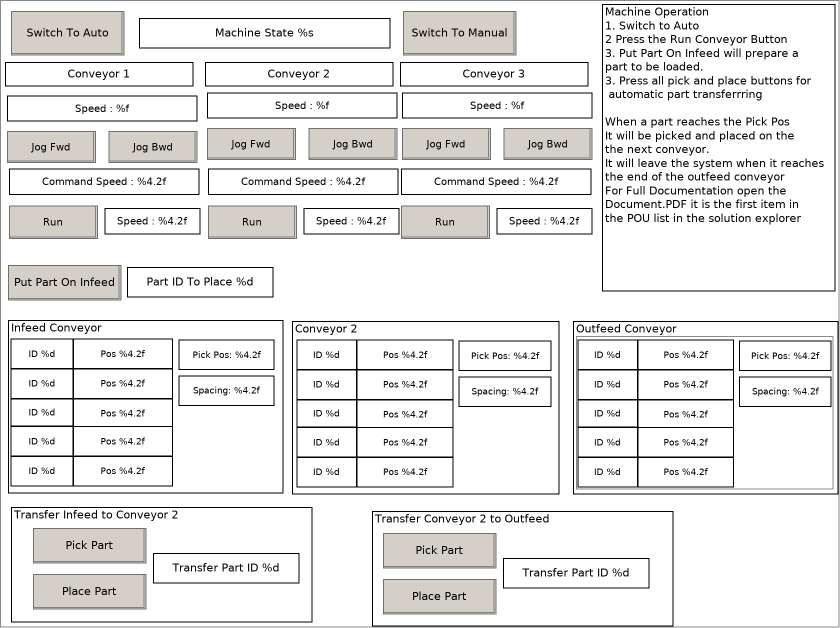
VISUALIZATION V_OOP_Conveyor  // 840x628
    Group (11,507 301x115)
        Rectangle (0,0 301x115), "Transfer Infeed to Conveyor 2"
        Button (22,21 113x35), "Pick Part", pressed state: MAIN.fbOOPConveyor.bPickPart
            toggle MAIN.fbOOPConveyor.bPickPart
        Rectangle (142,46 146x30), "Transfer Part ID %d", text variable: MAIN.fbOOPConveyor.fbTransfer1.stPart.iIDNumber
        Button (22,67 113x35), "Place Part", pressed state: MAIN.fbOOPConveyor.bPlacePart
            toggle MAIN.fbOOPConveyor.bPlacePart
    Button (11,11 113x44), "Switch To Auto"
        OnMouseDown: execute { MAIN.fbOOPConveyor.eMachineState := E_SwitchingToAuto; }
    Button (403,11 113x44), "Switch To Manual"
        OnMouseDown: execute { MAIN.fbOOPConveyor.eMachineState := E_SwitchingToManual; }
    Rectangle (139,18 251x30), "Machine State %s", text variable: MAIN.fbOOPConveyor.eMachineState
    Frame (10,99 189x66)
        shows Conveyor(bJogFwd := MAIN.fbOOPConveyor.bJogFwd, bJogBwd := MAIN.fbOOPConveyor.bJogBwd, fSpeed := MAIN.fbOOPConveyor.AxisRef[1].NcToPlc.ActVelo)
    Rectangle (5,62 188x24), "Conveyor 1"
    Frame (210,96 189x66)
        shows Conveyor(bJogFwd := MAIN.fbOOPConveyor.bJogFwd, bJogBwd := MAIN.fbOOPConveyor.bJogBwd, fSpeed := MAIN.fbOOPConveyor.iAnalogValue)
    Rectangle (205,62 188x24), "Conveyor 2"
    Frame (405,96 189x66)
        shows Conveyor(bJogFwd := MAIN.fbOOPConveyor.bJogFwd, bJogBwd := MAIN.fbOOPConveyor.bJogBwd, fSpeed := MAIN.fbOOPConveyor.AxisRef[2].NcToPlc.ActVelo)
    Rectangle (400,62 188x24), "Conveyor 3"
    Frame (11,174 191x67)
        shows ConveyorAuto(bRunConveyor := MAIN.fbOOPConveyor.bRunConveyor, fActualSpeed := MAIN.fbOOPConveyor.AxisRef[1].NcToPlc.ActVelo, fCmdSpeed := MAIN.fbOOPConveyor.fConveyorCmdSpeed)
    Button (8,265 113x35), "Put Part On Infeed", pressed state: MAIN.fbOOPConveyor.bPartPresent
        toggle MAIN.fbOOPConveyor.bPartPresent
    Frame (210,174 191x67)
        shows ConveyorAuto(bRunConveyor := MAIN.fbOOPConveyor.bRunConveyor, fActualSpeed := MAIN.fbOOPConveyor.fbConveyor2.fCurrentSpeed, fCmdSpeed := MAIN.fbOOPConveyor.fConveyorCmdSpeed)
    Rectangle (127,267 146x30), "Part ID To Place %d", text variable: arrParts[1].iIDNumber
    Group (292,321 267x173)
        Rectangle (0,0 267x173), "Conveyor 2"
        Frame (3,15 258x153)
            shows ConveyorData(fbConveyor := MAIN.fbOOPConveyor.fbConveyor2)
    Frame (403,174 191x67)
        shows ConveyorAuto(bRunConveyor := MAIN.fbOOPConveyor.bRunConveyor, fActualSpeed := MAIN.fbOOPConveyor.fbConveyor3.fCurrentSpeed, fCmdSpeed := MAIN.fbOOPConveyor.fConveyorCmdSpeed)
    Rectangle (8,320 275x173), "Infeed Conveyor"
    Frame (9,335 267x153)
        shows ConveyorData(fbConveyor := MAIN.fbOOPConveyor.fbInfeedConveyor)
    Group (372,511 301x115)
        Rectangle (0,0 301x115), "Transfer Conveyor 2 to Outfeed"
        Button (11,22 113x35), "Pick Part", pressed state: MAIN.fbOOPConveyor.bPickPart2
            toggle MAIN.fbOOPConveyor.bPickPart2
        Rectangle (131,47 146x30), "Transfer Part ID %d", text variable: MAIN.fbOOPConveyor.fbTransfer2.stPart.iIDNumber
        Button (11,68 113x35), "Place Part", pressed state: MAIN.fbOOPConveyor.bPlacePart2
            toggle MAIN.fbOOPConveyor.bPlacePart2
    Group (573,321 265x173)
        Rectangle (0,0 265x173), "Outfeed Conveyor"
        Frame (3,15 257x153)
            shows ConveyorData(fbConveyor := MAIN.fbOOPConveyor.fbConveyor3)
    Rectangle (602,4 233x287), "Machine Operation 1. Switch to Auto 2 Press the Run Conveyor Button 3. Put Part On Infeed will prepare a part to be loaded. 3. Press all pick and place buttons for automatic part transferrring When a part reaches the Pick Pos It will be picked and placed on the the next conveyor. It will leave the system when it reaches the end of the outfeed conveyor For Full Documentation open the Document.PDF it is the first item in the POU list in the solution explorer"
END_VISUALIZATION

// ---- POUs/Sample UML SC/Visu_Composite.TcVIS
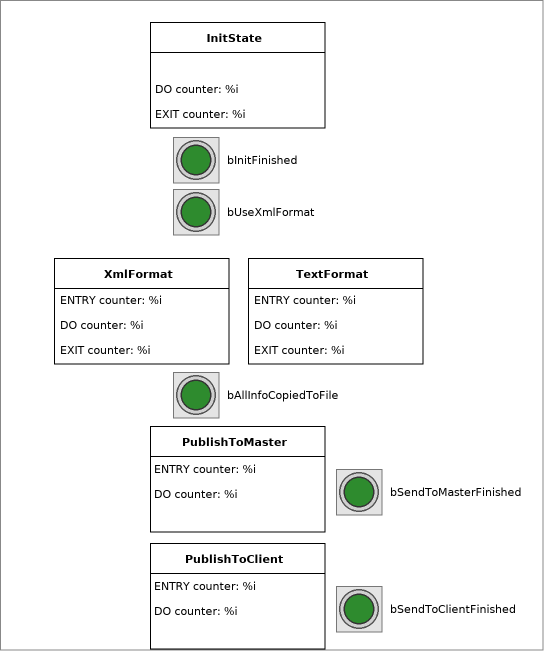
VISUALIZATION Visu_Composite  // 544x651
    Rectangle (150,22 175x106)
    Line (150,52) (325,52)
    Label (152,27 165x23), "InitState"
    Rectangle (54,258 175x106)
    Line (54,288) (229,288)
    Label (56,263 165x23), "XmlFormat"
    Rectangle (248,258 175x106)
    Line (248,288) (423,288)
    Label (250,263 165x23), "TextFormat"
    Rectangle (150,426 175x106)
    Line (150,456) (325,456)
    Label (152,431 165x23), "PublishToMaster"
    Rectangle (150,543 175x106)
    Line (150,573) (325,573)
    Label (152,548 165x23), "PublishToClient"
    PushSwitch (173,137 46x46), variable: MAIN.fbUmlSc.bInitFinished, behaviour: TOGGLE, style: Switch-PushSwitch-Green
    Label (224,149 118x23), "bInitFinished"
    PushSwitch (173,189 46x46), variable: MAIN.fbUmlSc.bUseXmlFormat, behaviour: TOGGLE, style: Switch-PushSwitch-Green
    Label (224,201 118x23), "bUseXmlFormat"
    PushSwitch (173,372 46x46), variable: MAIN.fbUmlSc.bAllInfoCopiedToFile, behaviour: TOGGLE, style: Switch-PushSwitch-Green
    Label (224,384 137x23), "bAllInfoCopiedToFile"
    PushSwitch (336,469 46x46), variable: MAIN.fbUmlSc.bSendToMasterFinished, behaviour: TOGGLE, style: Switch-PushSwitch-Green
    Label (387,481 155x23), "bSendToMasterFinished"
    PushSwitch (336,586 46x46), variable: MAIN.fbUmlSc.bSendToClientFinished, behaviour: TOGGLE, style: Switch-PushSwitch-Green
    Label (387,598 141x23), "bSendToClientFinished"
    Rectangle (152,54 169x21), text variable: GVL.nCounterInit
    Rectangle (152,79 169x21), "DO counter: %i", text variable: GVL.nCounterInit
    Rectangle (152,104 169x21), "EXIT counter: %i", text variable: GVL.nCounterSaveInitSettings
    Rectangle (57,290 169x21), "ENTRY counter: %i", text variable: GVL.nCounterClearXml
    Rectangle (57,315 169x21), "DO counter: %i", text variable: GVL.nCounterFillXml
    Rectangle (57,340 169x21), "EXIT counter: %i", text variable: GVL.nCounterSaveXml
    Rectangle (251,290 169x21), "ENTRY counter: %i", text variable: GVL.nCounterClearText
    Rectangle (251,315 169x21), "DO counter: %i", text variable: GVL.nCounterFillText
    Rectangle (251,340 169x21), "EXIT counter: %i", text variable: GVL.nCounterSaveText
    Rectangle (151,459 169x21), "ENTRY counter: %i", text variable: GVL.nCounterGetMasterID
    Rectangle (151,484 169x21), "DO counter: %i", text variable: GVL.nCounterSendToMaster
    Rectangle (151,509 169x21), text variable: GVL.nCounterInit
    Rectangle (151,576 169x21), "ENTRY counter: %i", text variable: GVL.nCounterGetClientID
    Rectangle (151,601 169x21), "DO counter: %i", text variable: GVL.nCounterSendToClient
    Rectangle (151,626 169x21), text variable: GVL.nCounterInit
END_VISUALIZATION

// ---- POUs/Sample UML SC/Visu_Lamp.TcVIS
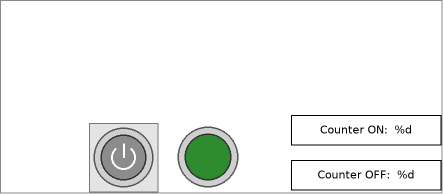
VISUALIZATION Visu_Lamp  // 443x194
    Lamp1 (173,122 70x70), variable: MAIN.fbUmlSc_Lamp.ObLamp, style: Lamp-Lamp1-Green
    PowerSwitch (69,123 109x69), variable: MAIN.fbUmlSc_Lamp.bPower, behaviour: TOGGLE, style: Switch-PowerSwitch-Gray
    Rectangle (291,115 150x30), "Counter ON: %d", text variable: MAIN.fbUmlSc_Lamp.nCounterOn
    Rectangle (291,160 150x30), "Counter OFF: %d", text variable: MAIN.fbUmlSc_Lamp.nCounterOff
END_VISUALIZATION

// ---- VISUs/MotionProfiles.TcVIS
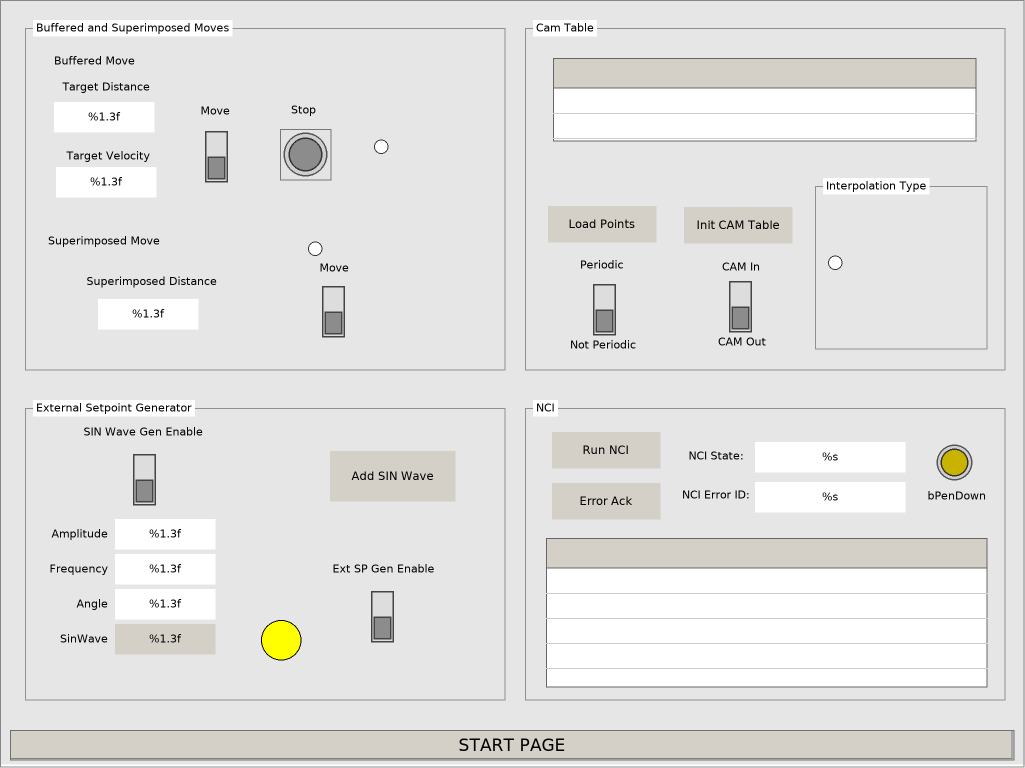
VISUALIZATION MotionProfiles  // 1025x768
    Rectangle (1,-4 1024x768)
    Button (10,730 1004x30), "START PAGE"
        OnMouseClick: change screen: HmiStartPage
    GroupBox (25,20 480x350), "Buffered and Superimposed Moves"
        Ellipse (236,600 40x40), colour toggle: Ext_SP_Gen.bAddSin
            toggle Ext_SP_Gen.bAddSin
        Label (12,30 115x22), "Buffered Move"
        Rectangle (29,82 100x30), "%1.3f", text variable: Axis3.lrMstrTarg2
            OnMouseDown: write the text variable via VisuDialogs.Numpad
        Rectangle (31,147 100x30), "%1.3f", text variable: Axis3.lrMstrVelo2
            OnMouseDown: write the text variable via VisuDialogs.Numpad
        Rectangle (30,56 98x22), "Target Distance"
        Rectangle (30,125 98x22), "Target Velocity"
        DipSwitch (166,108 51x57), variable: Axis3.bMvMstr2, behaviour: TOGGLE, style: Switch-DipSwitch-Gray
        RadioButton (347,95 96x63), variable: Axis3.iMstrMvMode2
            Areas[0]: Text=Absolute
            Areas[1]: Text=Relative
        PushSwitch (255,106 51x57), variable: Axis3.bStop, behaviour: TOGGLE, style: Switch-PushSwitch-Gray
        Label (12,210 134x22), "Superimposed Move"
        Label (159,80 63x22), "Move"
        Label (247,79 63x22), "Stop"
        Rectangle (73,279 100x30), "%1.3f", text variable: Axis3.lrMstrTarg3
            OnMouseDown: write the text variable via VisuDialogs.Numpad
        Rectangle (53,251 142x21), "Superimposed Distance"
        DipSwitch (283,263 51x57), variable: Axis3.bMvMstr2, behaviour: TOGGLE, style: Switch-DipSwitch-Gray
        Label (278,237 63x22), "Move"
    GroupBox (25,400 480x300), "External Setpoint Generator"
        DipSwitch (94,51 51x57), variable: Ext_SP_Gen.bSinGen, behaviour: TOGGLE, style: Switch-DipSwitch-Gray
        Label (45,21 147x22), "SIN Wave Gen Enable"
        DipSwitch (332,188 51x57), variable: Ext_SP_Gen.bMstrExtSP, behaviour: TOGGLE, style: Switch-DipSwitch-Gray
        Label (285,154 147x30), "Ext SP Gen Enable"
        Rectangle (11,158 75x22), "Frequency"
        Rectangle (305,51 125x50), "Add SIN Wave", colour toggle: Ext_SP_Gen.bAddSin
            toggle Ext_SP_Gen.bAddSin p2164770859=TRUE
    GroupBox (525,400 480x300), "NCI"
        Table (21,138 441x149), data array: NCI.aGCodeLines
            p3854506369: NCI.aGCodeLines[INDEX]
            p2232123230: Last 5 executed Gcode blocks
        Label (150,41 82x30), "NCI State:"
        Lamp1 (409,41 41x43), variable: NCI.bPenDown, style: Lamp-Lamp1-Yellow
        Rectangle (230,42 150x30), "%s", text variable: NCI.nNCI_State
        Label (150,80 82x30), "NCI Error ID:"
        Rectangle (230,82 150x30), "%s", text variable: NCI.nNciErrId
        Rectangle (27,32 108x36), "Run NCI", colour toggle: bRevSeqStart
            tap NCI.bRunNCI
        Rectangle (27,83 108x36), "Error Ack", colour toggle: bRevSeqStart
            tap NCI.bErrorAck
        Label (386,80 92x32), "bPenDown"
    GroupBox (525,20 480x350), "Cam Table"
        Rectangle (23,186 108x36), "Load Points", colour toggle: bRevSeqStart
            tap CamTable.bLoadPoints
        Rectangle (159,187 108x36), "Init CAM Table", colour toggle: bRevSeqStart
            tap CamTable.bCamInit
        DipSwitch (190,258 51x57), variable: CamTable.bCamIn, behaviour: TOGGLE, style: Switch-DipSwitch-Gray
        DipSwitch (54,261 51x57), variable: CamTable.bPeriodic, input disabled if: CamTable.bCamIn, behaviour: TOGGLE, style: Switch-DipSwitch-Gray
        Rectangle (168,311 98x22), "CAM Out"
        Rectangle (167,236 98x22), "CAM In"
        Rectangle (29,314 98x22), "Not Periodic"
        Rectangle (28,234 98x22), "Periodic"
        Table (28,38 423x83), data array: CamTable.arCamTable
            p3854506369: CamTable.arCamTable[0,INDEX]
            p1892666644: CamTable.arCamTable[1,INDEX]
            p338671338: CamTable.arCamTable[2,INDEX]
            p2170511999: CamTable.arCamTable[3,INDEX]
            p3723444502: CamTable.arCamTable[4,INDEX]
            p1218418051: CamTable.arCamTable[5,INDEX]
            p746581629: CamMotnFns.CamMotnFnPts[INDEX].SlavePos
            p3104783080: CamMotnFns.CamMotnFnPts[INDEX].SlaveVelo
            p2501879983: CamMotnFns.CamMotnFnPts[INDEX].SlaveAcc
            p7306298: CamMotnFns.CamMotnFnPts[INDEX].SlaveJerk
            p1137915858: CamTable.iSelY
            p1420305297: CamTable.iSelX
        GroupBox (290,158 172x171), "Interpolation Type"
            RadioButton (-509,19 137x103), variable: CamTable.iInterpType, input disabled if: CamTable.bCamIn
                Areas[0]: Text=Linear
                Areas[1]: Text=Spline
                Areas[2]: Text=Sliding Spline
        RadioButton (301,184 150x117), variable: CamTable.iInterpType, input disabled if: CamTable.bCamIn
            Areas[0]: Text=Linear
            Areas[1]: Text=Spline
            Areas[2]: Text=Sliding Spline
    Rectangle (115,624 100x30), "%1.3f", text variable: Ext_SP_Gen.lrSinWave
    Rectangle (115,589 100x30), "%1.3f", text variable: Ext_SP_Gen.rDeg
        OnMouseDown: write the text variable via VisuDialogs.Numpad
    Rectangle (58,593 53x22), "Angle"
    Rectangle (37,628 74x22), "SinWave"
    Rectangle (115,519 100x30), "%1.3f", text variable: Ext_SP_Gen.rSinAmp
        OnMouseDown: write the text variable via VisuDialogs.Numpad
    Rectangle (38,523 73x22), "Amplitude"
    Rectangle (115,554 100x30), "%1.3f", text variable: Ext_SP_Gen.rDegStep
        OnMouseDown: write the text variable via VisuDialogs.Numpad
END_VISUALIZATION

// ---- VISUs/HmiEtherCatDiagnostic.TcVIS
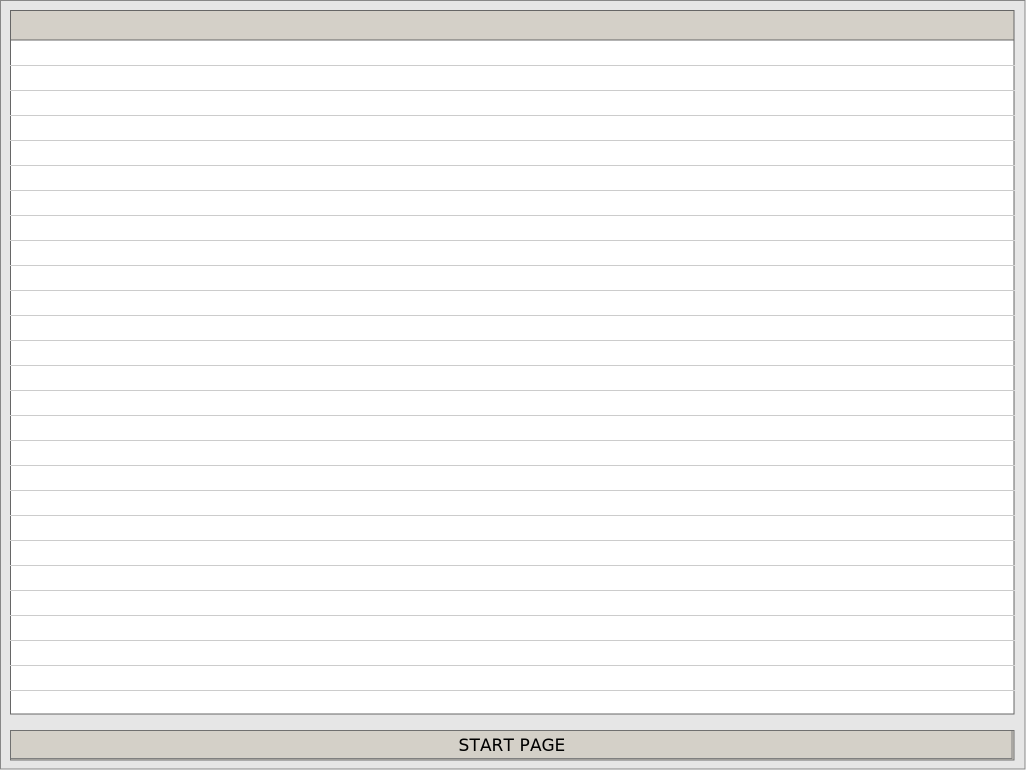
VISUALIZATION HmiEtherCatDiagnostic  // 1026x770
    Rectangle (0,0 1024x768)
    Button (10,730 1004x30), "START PAGE"
        OnMouseClick: change screen: HmiStartPage
    Table (10,10 1004x704), data array: fbDiagnosticEtherCAT.stEcTerminalDiagInfo
        p3854506369: fbDiagnosticEtherCAT.stEcTerminalDiagInfo[INDEX].nAddr
        p1892666644: fbDiagnosticEtherCAT.stEcTerminalDiagInfo[INDEX].sType
        p338671338: fbDiagnosticEtherCAT.stEcTerminalDiagInfo[INDEX].sName
        p2170511999: fbDiagnosticEtherCAT.stEcTerminalDiagInfo[INDEX].sTerminalStatus
END_VISUALIZATION

// ---- VISUs/HmiAxisReversingSequence.TcVIS
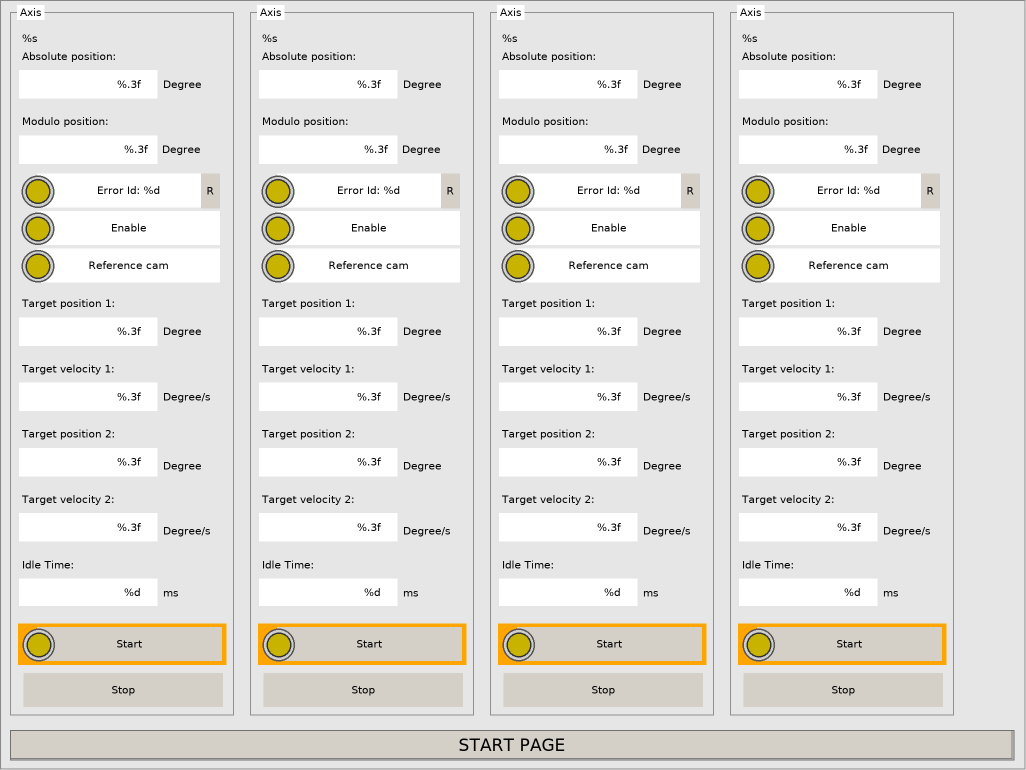
VISUALIZATION HmiAxisReversingSequence  // 1026x770
    Rectangle (0,0 1024x768)
    Button (10,730 1004x30), "START PAGE"
        OnMouseClick: change screen: HmiStartPage
    Frame (10,5 230x710)
        shows TplAxisReversingSequence(sAxisDescription := Axis1.sAxisDescription, fAbsolutePositon := stAxis1.NcToPlc.ActPos, fModuloPositon := stAxis1.NcToPlc.ModuloActPos, bError := Axis1.bAxisErr, nErrorId := Axis1.nAxisErrId, bReset := Axis1.bReset, bPowerStatus := Axis1.fbAxis.bPowerStatus, bReferenceCam := bStepperReferenceCam, bRevSeqStart := Axis1.bRevSeqStart, bRevSeqStop := Axis1.fbAxis.bRevSeqStop, fRevSeqTargetPos1 := Axis1.fbAxis.fRevSeqTargetPos1, fRevSeqTargetVelo1 := Axis1.fbAxis.fRevSeqTargetVelo1, fRevSeqTargetPos2 := Axis1.fbAxis.fRevSeqTargetPos2, fRevSeqTargetVelo2 := Axis1.fbAxis.fRevSeqTargetVelo2, nRevSeqIdleTime := Axis1.fbAxis.nRevSeqIdleTime, bRevSeqDone := Axis1.fbAxis.bRevSeqDone, bRevSeqBusy := Axis1.fbAxis.bRevSeqBusy)
    Frame (250,5 230x710)
        shows TplAxisReversingSequence(sAxisDescription := Axis2.sAxisDescription, fAbsolutePositon := stAxis2.NcToPlc.ActPos, fModuloPositon := stAxis2.NcToPlc.ModuloActPos, bError := Axis2.bAxisErr, nErrorId := Axis2.nAxisErrId, bReset := Axis2.bReset, bPowerStatus := Axis2.fbAxis.bPowerStatus, bReferenceCam := bAxis2ReferenceCamEL7, bRevSeqStart := Axis2.bRevSeqStart, bRevSeqStop := Axis2.fbAxis.bRevSeqStop, fRevSeqTargetPos1 := Axis2.fbAxis.fRevSeqTargetPos1, fRevSeqTargetVelo1 := Axis2.fbAxis.fRevSeqTargetVelo1, fRevSeqTargetPos2 := Axis2.fbAxis.fRevSeqTargetPos2, fRevSeqTargetVelo2 := Axis2.fbAxis.fRevSeqTargetVelo2, nRevSeqIdleTime := Axis2.fbAxis.nRevSeqIdleTime, bRevSeqDone := Axis2.fbAxis.bRevSeqDone, bRevSeqBusy := Axis2.fbAxis.bRevSeqBusy)
    Frame (490,5 230x710)
        shows TplAxisReversingSequence(sAxisDescription := Axis3.sAxisDescription, fAbsolutePositon := stAxis3.NcToPlc.ActPos, fModuloPositon := stAxis3.NcToPlc.ModuloActPos, bError := Axis3.bAxisErr, nErrorId := Axis3.nAxisErrId, bReset := Axis3.bReset, bPowerStatus := Axis3.fbAxis.bPowerStatus, bReferenceCam := AxisGeneral.bAxis3ReferenceCam, bRevSeqStart := Axis3.bRevSeqStart, bRevSeqStop := Axis3.fbAxis.bRevSeqStop, fRevSeqTargetPos1 := Axis3.fbAxis.fRevSeqTargetPos1, fRevSeqTargetVelo1 := Axis3.fbAxis.fRevSeqTargetVelo1, fRevSeqTargetPos2 := Axis3.fbAxis.fRevSeqTargetPos2, fRevSeqTargetVelo2 := Axis3.fbAxis.fRevSeqTargetVelo2, nRevSeqIdleTime := Axis3.fbAxis.nRevSeqIdleTime, bRevSeqDone := Axis3.fbAxis.bRevSeqDone, bRevSeqBusy := Axis3.fbAxis.bRevSeqBusy)
    Frame (730,5 230x710)
        shows TplAxisReversingSequence(sAxisDescription := Axis4.sAxisDescription, fAbsolutePositon := stAxis4.NcToPlc.ActPos, fModuloPositon := stAxis4.NcToPlc.ModuloActPos, bError := Axis4.bAxisErr, nErrorId := Axis4.nAxisErrId, bReset := Axis4.bReset, bPowerStatus := Axis4.fbAxis.bPowerStatus, bReferenceCam := AxisGeneral.bAxis4ReferenceCam, bRevSeqStart := Axis4.bRevSeqStart, bRevSeqStop := Axis4.fbAxis.bRevSeqStop, fRevSeqTargetPos1 := Axis4.fbAxis.fRevSeqTargetPos1, fRevSeqTargetVelo1 := Axis4.fbAxis.fRevSeqTargetVelo1, fRevSeqTargetPos2 := Axis4.fbAxis.fRevSeqTargetPos2, fRevSeqTargetVelo2 := Axis4.fbAxis.fRevSeqTargetVelo2, nRevSeqIdleTime := Axis4.fbAxis.nRevSeqIdleTime, bRevSeqDone := Axis4.fbAxis.bRevSeqDone, bRevSeqBusy := Axis4.fbAxis.bRevSeqBusy)
END_VISUALIZATION

// ---- VISUs/HmiStartPage.TcVIS
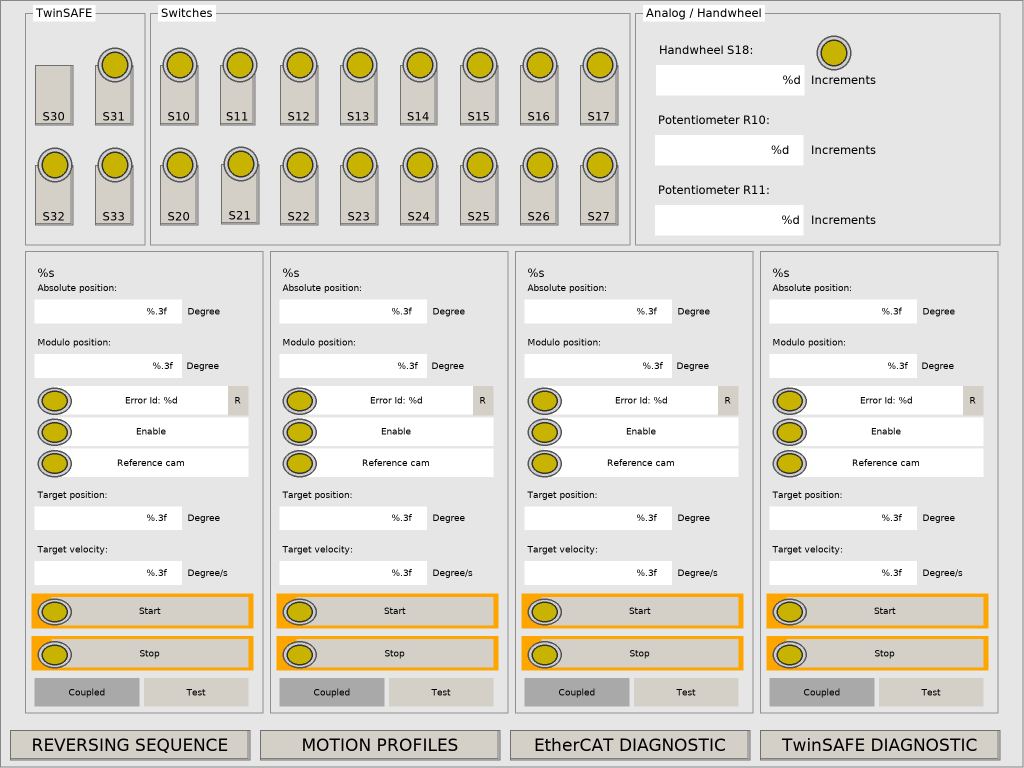
VISUALIZATION HmiStartPage  // 1024x768
    Rectangle (0,0 1024x768)
    Button (760,730 240x30), "TwinSAFE DIAGNOSTIC"
        OnMouseClick: change screen: HmiTwinSAFEDiagnostic
    Button (510,730 240x30), "EtherCAT DIAGNOSTIC"
        OnMouseClick: change screen: HmiEtherCatDiagnostic
    GroupBox (25,5 120x240), "TwinSAFE"
        Button (10,60 38x60), "S30", colour toggle: NOT TwinSAFE.fbSafeConnectionEL1904_1_Group1.bChannel1 and NOT TwinSAFE.fbSafeConnectionEL1904_1_Group1.bChannel2
            toggle bSwitchS31
        Button (70,60 38x60), "S31", colour toggle: bSwitchS31
            toggle bSwitchS31
        Lamp1 (70,40 40x40), variable: bLedH31, style: Lamp-Lamp1-Yellow
        Button (70,160 38x60), "S33", colour toggle: NOT TwinSAFE.fbSafeConnectionEL1904_2_Group1.bChannel3 and TwinSAFE.fbSafeConnectionEL1904_2_Group1.bChannel4
            toggle bSwitchS31
        Lamp1 (70,140 40x40), variable: bLedH33, style: Lamp-Lamp1-Yellow
        Button (10,160 38x60), "S32", colour toggle: NOT TwinSAFE.fbSafeConnectionEL1904_2_Group1.bChannel1 and NOT TwinSAFE.fbSafeConnectionEL1904_2_Group1.bChannel2
            toggle bSwitchS31
        Lamp1 (10,140 40x40), variable: bLedH32, style: Lamp-Lamp1-Yellow
    GroupBox (150,5 480x240), "Switches"
        Button (10,60 38x60), "S10", colour toggle: bSwitchS10
            toggle bSwitchS10
        Lamp1 (10,40 40x40), variable: bLedH10, style: Lamp-Lamp1-Yellow
        Button (70,60 35x60), "S11", colour toggle: bSwitchS11
            toggle bSwitchS11
        Lamp1 (70,40 40x40), variable: bLedH11, style: Lamp-Lamp1-Yellow
        Button (130,60 38x60), "S12", colour toggle: bSwitchS12
            toggle bSwitchS12
        Lamp1 (130,40 40x40), variable: bLedH12, style: Lamp-Lamp1-Yellow
        Button (190,60 37x60), "S13", colour toggle: bSwitchS13
            toggle bSwitchS13
        Lamp1 (190,40 40x40), variable: bLedH13, style: Lamp-Lamp1-Yellow
        Button (250,60 37x60), "S14", colour toggle: bSwitchS14
            toggle bSwitchS14
        Lamp1 (250,40 40x40), variable: bLedH14, style: Lamp-Lamp1-Yellow
        Button (310,60 38x60), "S15", colour toggle: bSwitchS15
            toggle bSwitchS15
        Lamp1 (310,40 40x40), variable: bLedH15, style: Lamp-Lamp1-Yellow
        Button (370,60 38x60), "S16", colour toggle: bSwitchS16
            toggle bSwitchS16
        Lamp1 (370,40 40x40), variable: bLedH16, style: Lamp-Lamp1-Yellow
        Button (430,60 38x60), "S17", colour toggle: bSwitchS17
            toggle bSwitchS17
        Lamp1 (430,40 40x40), variable: bLedH17, style: Lamp-Lamp1-Yellow
        Button (10,160 38x60), "S20", colour toggle: bSwitchS20
            toggle bSwitchS20
        Lamp1 (10,140 40x40), variable: bLedH20, style: Lamp-Lamp1-Yellow
        Button (71,159 38x60), "S21", colour toggle: bSwitchS21
            toggle bSwitchS21
        Lamp1 (71,139 40x40), variable: bLedH21, style: Lamp-Lamp1-Yellow
        Button (130,160 38x60), "S22", colour toggle: bSwitchS22
            toggle bSwitchS22
        Lamp1 (130,140 40x40), variable: bLedH22, style: Lamp-Lamp1-Yellow
        Button (190,160 38x60), "S23", colour toggle: bSwitchS23
            toggle bSwitchS23
        Lamp1 (190,140 40x40), variable: bLedH23, style: Lamp-Lamp1-Yellow
        Button (250,160 38x60), "S24", colour toggle: bSwitchS24
            toggle bSwitchS24
        Lamp1 (250,140 40x40), variable: bLedH24, style: Lamp-Lamp1-Yellow
        Button (310,160 38x60), "S25", colour toggle: bSwitchS25
            toggle bSwitchS25
        Lamp1 (310,140 40x40), variable: bLedH25, style: Lamp-Lamp1-Yellow
        Button (370,160 38x60), "S26", colour toggle: nAX5203DigitalInputs.2
            toggle nAX5203DigitalInputs.2
        Lamp1 (370,140 40x40), variable: bLedH26, style: Lamp-Lamp1-Yellow
        Button (430,160 38x60), "S27", colour toggle: nAX5203DigitalInputs.3
            toggle nAX5203DigitalInputs.3
        Lamp1 (430,140 40x40), variable: nAX5203DigitalOutputs.7, style: Lamp-Lamp1-Yellow
    GroupBox (635,5 365x240), "Analog / Handwheel"
        Rectangle (20,200 148x30), "%d", text variable: aOsAnalogInR11[0]
            OnMouseClick: write the text variable via VisuDialogs.Numpad, min 0, max 32767
        Label (173,200 118x30), "Increments"
        Label (20,170 197x30), "Potentiometer R11:"
        Rectangle (20,130 148x30), "%d", text variable: nAnalogInR10
            OnMouseClick: write the text variable via VisuDialogs.Numpad, min 0, max 32767
        Label (173,130 121x30), "Increments"
        Label (20,100 216x30), "Potentiometer R10:"
        Lamp1 (179,28 40x40), variable: bHandwheelSwitchS28, style: Lamp-Lamp1-Yellow
        Rectangle (21,60 148x30), "%d", text variable: nHandwheelCounter
            OnMouseClick: write the text variable via VisuDialogs.Numpad
        Label (173,60 133x30), "Increments"
        Label (21,30 216x30), "Handwheel S18:"
    Frame (25,245 240x470)
        shows TplAxisControl(sAxisDescription := Axis1.sAxisDescription, fAbsolutePositon := stAxis1.NcToPlc.ActPos, fModuloPositon := stAxis1.NcToPlc.ModuloActPos, bError := Axis1.bAxisErr, nErrorId := Axis1.nAxisErrId, bReset := Axis1.bReset, bPowerStatus := Axis1.fbAxis.bPowerStatus, bReferenceCam := bStepperReferenceCam, fMoveAbsPosition := Axis1.fMoveAbsPosition, fMoveAbsVelocity := Axis1.fMoveAbsVelocity, bStartMoveAbs := Axis1.bStartMoveAbs, bMoveAbsBusy := Axis1.bMoveAbsBusy, bMoveAbsDone := Axis1.bMoveAbsDone, bStop := Axis1.bStop, bStopBusy := Axis1.bStopAxisBusy, bStopDone := Axis1.bStopAxisDone, bAxisCoupled := Axis1.bAxisCoupled, bTestChangeTargetPosAxis := Axis1.bTestChangeTargetPos)
    Frame (270,245 240x470)
        shows TplAxisControl(sAxisDescription := Axis2.sAxisDescription, fAbsolutePositon := stAxis2.NcToPlc.ActPos, fModuloPositon := stAxis2.NcToPlc.ModuloActPos, bError := Axis2.bAxisErr, nErrorId := Axis2.nAxisErrId, bReset := Axis2.bReset, bPowerStatus := Axis2.fbAxis.bPowerStatus, bReferenceCam := bAxis2ReferenceCamEL7, fMoveAbsPosition := Axis2.fMoveAbsPosition, fMoveAbsVelocity := Axis2.fMoveAbsVelocity, bStartMoveAbs := Axis2.bStartMoveAbs, bMoveAbsBusy := Axis2.bMoveAbsBusy, bMoveAbsDone := Axis2.bMoveAbsDone, bStop := Axis2.bStop, bStopBusy := Axis2.bStopAxisBusy, bStopDone := Axis2.bStopAxisDone, bAxisCoupled := Axis2.bAxisCoupled, bTestChangeTargetPosAxis := Axis2.bTestChangeTargetPos)
    Frame (515,245 240x470)
        shows TplAxisControl(sAxisDescription := Axis3.sAxisDescription, fAbsolutePositon := stAxis3.NcToPlc.ActPos, fModuloPositon := stAxis3.NcToPlc.ModuloActPos, bError := Axis3.bAxisErr, nErrorId := Axis3.nAxisErrId, bReset := Axis3.bReset, bPowerStatus := Axis3.fbAxis.bPowerStatus, bReferenceCam := AxisGeneral.bAxis3ReferenceCam, fMoveAbsPosition := Axis3.fMoveAbsPosition, fMoveAbsVelocity := Axis3.fMoveAbsVelocity, bStartMoveAbs := Axis3.bStartMoveAbs, bMoveAbsBusy := Axis3.bMoveAbsBusy, bMoveAbsDone := Axis3.bMoveAbsDone, bStop := Axis3.bStop, bStopBusy := Axis3.bStopAxisBusy, bStopDone := Axis3.bStopAxisDone, bAxisCoupled := Axis3.bAxisCoupled, bTestChangeTargetPosAxis := Axis3.bTestChangeTargetPos)
    Frame (760,245 240x470)
        shows TplAxisControl(sAxisDescription := Axis4.sAxisDescription, fAbsolutePositon := stAxis4.NcToPlc.ActPos, fModuloPositon := stAxis4.NcToPlc.ModuloActPos, bError := Axis4.bAxisErr, nErrorId := Axis4.nAxisErrId, bReset := Axis4.bReset, bPowerStatus := Axis4.fbAxis.bPowerStatus, bReferenceCam := AxisGeneral.bAxis4ReferenceCam, fMoveAbsPosition := Axis4.fMoveAbsPosition, fMoveAbsVelocity := Axis4.fMoveAbsVelocity, bStartMoveAbs := Axis4.bStartMoveAbs, bMoveAbsBusy := Axis4.bMoveAbsBusy, bMoveAbsDone := Axis4.bMoveAbsDone, bStop := Axis4.bStop, bStopBusy := Axis4.bStopAxisBusy, bStopDone := Axis4.bStopAxisDone, bAxisCoupled := Axis4.bAxisCoupled, bTestChangeTargetPosAxis := Axis4.bTestChangeTargetPos)
    Button (10,730 240x30), "REVERSING SEQUENCE"
        OnMouseClick: change screen: HmiAxisReversingSequence
    Button (260,730 240x30), "MOTION PROFILES"
        OnMouseClick: change screen: MotionProfiles
END_VISUALIZATION

// ---- VISUs/HmiTemplatesAxis/TplAxisControl.TcVIS
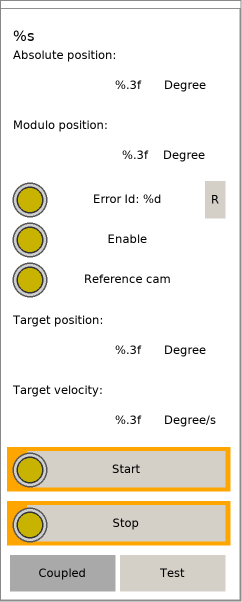
VISUALIZATION TplAxisControl  // 242x602
VAR_IN_OUT
	sAxisDescription				:STRING;
	fAbsolutePositon				:LREAL;
	fModuloPositon					:LREAL;
	bError							:BOOL;
	nErrorId						:DWORD;
	bReset							:BOOL;
	bPowerStatus					:BOOL;
	bReferenceCam					:BOOL;
	fMoveAbsPosition				:LREAL;
	fMoveAbsVelocity				:LREAL;
	bStartMoveAbs					:BOOL;
	bMoveAbsBusy					:BOOL;
	bMoveAbsDone					:BOOL;
	bStop							:BOOL;
	bStopBusy						:BOOL;
	bStopDone						:BOOL;
	bAxisCoupled					:BOOL;
	bTestChangeTargetPosAxis		:BOOL;
END_VAR
(* End *)
    GroupBox (0,0 240x600)
        Rectangle (7,501 223x44), invisible if: NOT bStopBusy
        Rectangle (7,447 223x44), invisible if: NOT bMoveAbsBusy
        Rectangle (27,451 198x36), "Start", colour toggle: bStartMoveAbs
            toggle bStartMoveAbs
        Group (10,110 230x60)
            Rectangle (0,30 148x30), "%.3f", text variable: fModuloPositon
            Label (150,30 80x30), "Degree"
            Label (0,0 200x30), "Modulo position:"
        Group (10,40 227x60)
            Rectangle (0,30 148x30), "%.3f", text variable: fAbsolutePositon
            Label (151,30 76x30), "Degree"
            Label (0,0 216x30), "Absolute position:"
        Group (10,180 200x40)
            Rectangle (20,1 195x36), "Error Id: %d", text variable: nErrorId
            Lamp1 (0,0 40x40), variable: bError, style: Lamp-Lamp1-Yellow
        Group (10,220 215x40)
            Rectangle (20,1 195x36), "Enable"
            Lamp1 (0,0 40x40), variable: bPowerStatus, style: Lamp-Lamp1-Yellow
        Group (10,260 215x40)
            Rectangle (20,1 195x36), "Reference cam"
            Lamp1 (0,0 40x40), variable: bReferenceCam, style: Lamp-Lamp1-Yellow
        Rectangle (205,181 20x37), "R", tooltip "Reset", colour toggle: bReset
            tap bReset
        Rectangle (27,505 198x36), "Stop", colour toggle: bStop
            toggle bStop
        Rectangle (10,555 105x36), "Coupled", colour toggle: bAxisCoupled
        Rectangle (10,25 230x22), "%s", text variable: sAxisDescription
        Rectangle (10,335 148x30), "%.3f", text variable: fMoveAbsPosition
            OnMouseClick: write the text variable via VisuDialogs.Numpad
        Label (161,335 76x30), "Degree"
        Label (10,305 216x30), "Target position:"
        Rectangle (10,405 148x30), "%.3f", text variable: fMoveAbsVelocity
            OnMouseClick: write the text variable via VisuDialogs.Numpad
        Label (161,405 76x30), "Degree/s"
        Label (10,375 216x30), "Target velocity:"
        Lamp1 (10,505 40x40), variable: bStopDone, style: Lamp-Lamp1-Yellow
        Rectangle (120,555 105x36), "Test", colour toggle: bTestChangeTargetPosAxis
            toggle bTestChangeTargetPosAxis
        Lamp1 (10,450 40x40), variable: bMoveAbsDone, style: Lamp-Lamp1-Yellow
END_VISUALIZATION

// ---- VISUs/HmiTemplatesAxis/TplAxisReversingSequence.TcVIS
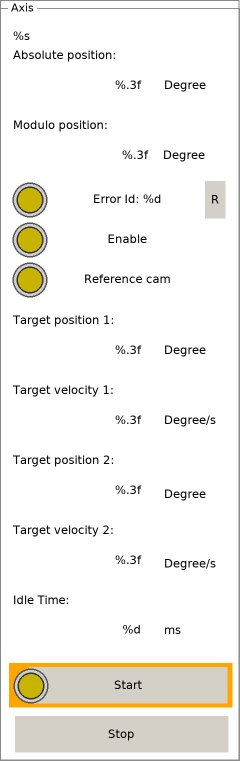
VISUALIZATION TplAxisReversingSequence  // 240x761
VAR_IN_OUT
	sAxisDescription				:STRING;
	fAbsolutePositon				:LREAL;
	fModuloPositon					:LREAL;
	bError							:BOOL;
	nErrorId						:DWORD;
	bReset							:BOOL;
	bPowerStatus					:BOOL;
	bReferenceCam					:BOOL;
	bRevSeqStart					:BOOL;
	bRevSeqStop						:BOOL;
	fRevSeqTargetPos1				:LREAL;
	fRevSeqTargetVelo1				:LREAL;
	fRevSeqTargetPos2				:LREAL;
	fRevSeqTargetVelo2				:LREAL;
	nRevSeqIdleTime					:UINT;
	bRevSeqDone						:BOOL;
	bRevSeqBusy						:BOOL;
END_VAR
    GroupBox (0,0 240x761), "Axis"
        Group (10,40 227x60)
            Rectangle (0,30 148x30), "%.3f", text variable: fAbsolutePositon
            Label (151,30 76x30), "Degree"
            Label (0,0 216x30), "Absolute position:"
        Group (10,180 200x40)
            Rectangle (20,1 195x36), "Error Id: %d", text variable: nErrorId
            Lamp1 (0,0 40x40), variable: bError, style: Lamp-Lamp1-Yellow
        Group (10,220 215x40)
            Rectangle (20,1 195x36), "Enable"
            Lamp1 (0,0 40x40), variable: bPowerStatus, style: Lamp-Lamp1-Yellow
        Group (10,260 215x40)
            Rectangle (20,1 195x36), "Reference cam"
            Lamp1 (0,0 40x40), variable: bReferenceCam, style: Lamp-Lamp1-Yellow
        Rectangle (205,181 20x37), "R", tooltip "Reset", colour toggle: bReset
            tap bReset
        Rectangle (10,25 230x22), "%s", text variable: sAxisDescription
        Rectangle (10,335 148x30), "%.3f", text variable: fRevSeqTargetPos1
            OnMouseClick: write the text variable via VisuDialogs.Numpad
        Label (161,335 76x30), "Degree"
        Label (10,305 216x30), "Target position 1:"
        Rectangle (10,405 148x30), "%.3f", text variable: fRevSeqTargetVelo1
            OnMouseClick: write the text variable via VisuDialogs.Numpad
        Label (161,405 76x30), "Degree/s"
        Group (10,110 230x60)
            Rectangle (0,30 148x30), "%.3f", text variable: fModuloPositon
            Label (150,30 80x30), "Degree"
            Label (0,0 200x30), "Modulo position:"
        Rectangle (9,663 223x44), invisible if: NOT bRevSeqBusy
        Rectangle (29,667 198x36), "Start", colour toggle: bRevSeqStart
            toggle bRevSeqStart
        Lamp1 (11,666 40x40), variable: bRevSeqDone, style: Lamp-Lamp1-Yellow
        Rectangle (15,716 213x36), "Stop", colour toggle: bRevSeqStop
            toggle bRevSeqStop
        Rectangle (10,615 148x29), "%d", text variable: nRevSeqIdleTime
            OnMouseClick: write the text variable via VisuDialogs.Numpad
        Label (10,585 216x30), "Idle Time:"
        Label (10,375 216x30), "Target velocity 1:"
    Label (161,479 76x30), "Degree"
    Rectangle (10,475 148x30), "%.3f", text variable: fRevSeqTargetPos2
        OnMouseClick: write the text variable via VisuDialogs.Numpad
    Label (10,445 216x30), "Target position 2:"
    Rectangle (10,545 148x30), "%.3f", text variable: fRevSeqTargetVelo2
        OnMouseClick: write the text variable via VisuDialogs.Numpad
    Label (161,549 76x29), "Degree/s"
    Label (10,515 216x30), "Target velocity 2:"
    Label (161,615 76x30), "ms"
END_VISUALIZATION

// ---- VISUs/HmiTemplatesTwinSAFE/TplTsConnectionAX5805.TcVIS
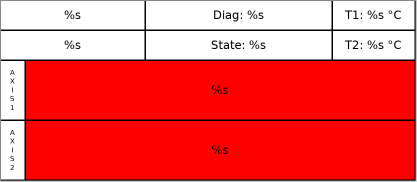
VISUALIZATION TplTsConnectionAX5805  // 417x182
VAR_IN_OUT
	stConnectionDiag 			:FB_TwinSafeConnectionAX5805;
END_VAR
(* End *)
    Rectangle (0,0 145x30), "%s", text variable: stConnectionDiag.sEcSlaveName
    Rectangle (25,60 49x30), "S-STO", colour toggle: stConnectionDiag.stSignalStatusMC1.bSafeTorqueOff_STO
    Rectangle (74,60 49x30), "S-SMM1", colour toggle: stConnectionDiag.stSignalStatusMC1.bSafeSpeedMonitor_SSM_1
    Rectangle (123,60 49x30), "S-SSM2", colour toggle: stConnectionDiag.stSignalStatusMC1.bSafeSpeedMonitor_SSM_2
    Rectangle (172,60 48x30), "S-SOS1", colour toggle: stConnectionDiag.stSignalStatusMC1.bSafeOperatingStop_SOS_1
    Rectangle (145,0 187x30), "Diag: %s", text variable: stConnectionDiag.sDiag, colour toggle: stConnectionDiag.sDiag <> 'No error'
    Rectangle (145,30 187x30), "State: %s", text variable: stConnectionDiag.sState
    Rectangle (0,30 145x30), "%s", text variable: stConnectionDiag.sEcSlaveType
    Rectangle (220,60 49x30), "S-SSR1", colour toggle: stConnectionDiag.stSignalStatusMC1.bSafeSpeedRange_SSR_1
    Rectangle (269,60 49x30), "S-SDIp", colour toggle: stConnectionDiag.stSignalStatusMC1.bSafeDirectionPositive_SDIp
    Rectangle (318,60 49x30), "S-SDIn", colour toggle: stConnectionDiag.stSignalStatusMC1.bSafeDirectionNegative_SDIn
    Rectangle (367,60 48x30), "S-Err Ack", colour toggle: stConnectionDiag.stSignalStatusMC1.bErrorAcknowledge_ErrAck
    Rectangle (25,90 49x30), "C-STO", colour toggle: stConnectionDiag.stSignalControlStatusMC1.bSafeTorqueOff_STO
    Rectangle (74,90 49x30), "C-SS1", colour toggle: stConnectionDiag.stSignalControlStatusMC1.bSafeStop1_SS1_1
    Rectangle (123,90 49x30), "C-SS2", colour toggle: stConnectionDiag.stSignalControlStatusMC1.bSafeStop2_SS2_1
    Rectangle (172,90 48x30), "C-SOS1", colour toggle: stConnectionDiag.stSignalControlStatusMC1.bSafeOperatingStop_SOS_1
    Rectangle (220,90 49x30), "C-SSR1", colour toggle: stConnectionDiag.stSignalControlStatusMC1.bSafeSpeedRange_SSR_1
    Rectangle (269,90 49x30), "C-SDIp", colour toggle: stConnectionDiag.stSignalControlStatusMC1.bSafeDirectionPositive_SDIp
    Rectangle (318,90 49x30), "C-SDIn", colour toggle: stConnectionDiag.stSignalControlStatusMC1.bSafeDirectionNegative_SDIn
    Rectangle (367,90 48x30), "C-Err Ack", colour toggle: stConnectionDiag.stSignalControlStatusMC1.bErrorAcknowledge_ErrAck
    Rectangle (332,0 83x30), "T1: %s °C", text variable: stConnectionDiag.stSlaveTemp.nInternalTemperature1, colour toggle: stConnectionDiag.bTempWarning
    Rectangle (332,30 83x30), "T2: %s °C", text variable: stConnectionDiag.stSlaveTemp.nInternalTemperature2, colour toggle: stConnectionDiag.bTempWarning
    Rectangle (25,120 49x30), "S-STO", colour toggle: stConnectionDiag.stSignalStatusMC2.bSafeTorqueOff_STO
    Rectangle (74,120 49x30), "S-SMM1", colour toggle: stConnectionDiag.stSignalStatusMC2.bSafeSpeedMonitor_SSM_1
    Rectangle (123,120 49x30), "S-SSM2", colour toggle: stConnectionDiag.stSignalStatusMC2.bSafeSpeedMonitor_SSM_2
    Rectangle (172,120 48x30), "S-SOS1", colour toggle: stConnectionDiag.stSignalStatusMC2.bSafeOperatingStop_SOS_1
    Rectangle (220,120 49x30), "S-SSR1", colour toggle: stConnectionDiag.stSignalStatusMC2.bSafeSpeedRange_SSR_1
    Rectangle (269,120 49x30), "S-SDIp", colour toggle: stConnectionDiag.stSignalStatusMC2.bSafeDirectionPositive_SDIp
    Rectangle (318,120 49x30), "S-SDIn", colour toggle: stConnectionDiag.stSignalStatusMC2.bSafeDirectionNegative_SDIn
    Rectangle (367,120 48x30), "S-Err Ack", colour toggle: stConnectionDiag.stSignalStatusMC2.bErrorAcknowledge_ErrAck
    Rectangle (25,150 49x30), "C-STO", colour toggle: stConnectionDiag.stSignalControlStatusMC2.bSafeTorqueOff_STO
    Rectangle (74,150 49x30), "C-SS1", colour toggle: stConnectionDiag.stSignalControlStatusMC2.bSafeStop1_SS1_1
    Rectangle (123,150 49x30), "C-SS2", colour toggle: stConnectionDiag.stSignalControlStatusMC2.bSafeStop2_SS2_1
    Rectangle (172,150 48x30), "C-SOS1", colour toggle: stConnectionDiag.stSignalControlStatusMC2.bSafeOperatingStop_SOS_1
    Rectangle (220,150 49x30), "C-SSR1", colour toggle: stConnectionDiag.stSignalControlStatusMC2.bSafeSpeedRange_SSR_1
    Rectangle (269,150 49x30), "C-SDIp", colour toggle: stConnectionDiag.stSignalControlStatusMC2.bSafeDirectionPositive_SDIp
    Rectangle (318,150 49x30), "C-SDIn", colour toggle: stConnectionDiag.stSignalControlStatusMC2.bSafeDirectionNegative_SDIn
    Rectangle (367,150 48x30), "C-Err Ack", colour toggle: stConnectionDiag.stSignalControlStatusMC2.bErrorAcknowledge_ErrAck
    Rectangle (0,60 25x60), "A X I S 1"
    Rectangle (0,120 25x60), "A X I S 2"
    Rectangle (26,61 388x58), "%s", text variable: stConnectionDiag.eErrIndicesFA82DiagnosisMC1, invisible if: NOT stConnectionDiag.bErrIndicesFA82DiagnosisMC1Err
    Rectangle (26,121 388x58), "%s", text variable: stConnectionDiag.eErrIndicesFA82DiagnosisMC2, invisible if: NOT stConnectionDiag.bErrIndicesFA82DiagnosisMC2Err
END_VISUALIZATION

// ---- VISUs/HmiTemplatesTwinSAFE/TplTsConnectionEK1914.TcVIS
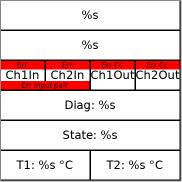
VISUALIZATION TplTsConnectionEK1914  // 182x182
VAR_IN_OUT
	stConnectionDiag 			:FB_TwinSafeConnectionEK1914;
END_VAR
(* End *)
    Rectangle (0,0 180x30), "%s", text variable: stConnectionDiag.sEcSlaveName, colour toggle: stConnectionDiag.sDiag = 'No error'
    Rectangle (0,60 45x30), "Ch1In", colour toggle: stConnectionDiag.bChannel1In
    Rectangle (45,60 45x30), "Ch2In", colour toggle: stConnectionDiag.bChannel2In
    Rectangle (90,60 45x30), "Ch1Out", colour toggle: stConnectionDiag.bChannel1Out
    Rectangle (135,60 45x30), "Ch2Out", colour toggle: stConnectionDiag.bChannel2Out
    Rectangle (0,90 180x30), "Diag: %s", text variable: stConnectionDiag.sDiag, colour toggle: stConnectionDiag.sDiag <> 'No error'
    Rectangle (0,120 180x30), "State: %s", text variable: stConnectionDiag.sState
    Rectangle (0,150 90x30), "T1: %s °C", text variable: stConnectionDiag.stSlaveTemp.nInternalTemperature1, colour toggle: stConnectionDiag.bTempWarning
    Rectangle (90,150 90x30), "T2: %s °C", text variable: stConnectionDiag.stSlaveTemp.nInternalTemperature2, colour toggle: stConnectionDiag.bTempWarning
    Rectangle (0,30 180x30), "%s", text variable: stConnectionDiag.sEcSlaveType
    Rectangle (1,61 43x8), "Err", invisible if: NOT stConnectionDiag.stTsDiagObjectsBitsEK1914.bErrInput1
    Rectangle (46,61 43x8), "Err", invisible if: NOT stConnectionDiag.stTsDiagObjectsBitsEK1914.bErrInput2
    Rectangle (91,61 43x8), "Err Cc", invisible if: NOT stConnectionDiag.stTsDiagObjectsBitsEK1914.bCcErrOutput1
    Rectangle (136,61 43x8), "Err Cc", invisible if: NOT stConnectionDiag.stTsDiagObjectsBitsEK1914.bCcErrOutput2
    Rectangle (1,81 88x8), "Err input pair", invisible if: NOT stConnectionDiag.stTsDiagObjectsBitsEK1914.bErrFirstInputPair
END_VISUALIZATION

// ---- VISUs/HmiTemplatesTwinSAFE/TplTsConnectionEL1904.TcVIS
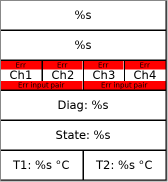
VISUALIZATION TplTsConnectionEL1904  // 168x182
VAR_IN_OUT
	stConnectionDiag 			:FB_TwinSafeConnectionEL1904;
END_VAR
(* End *)
    Rectangle (0,0 166x30), "%s", text variable: stConnectionDiag.sEcSlaveName, colour toggle: stConnectionDiag.sDiag = 'No error'
    Rectangle (0,60 42x30), "Ch1", colour toggle: stConnectionDiag.bChannel1
    Rectangle (42,60 42x30), "Ch2", colour toggle: stConnectionDiag.bChannel2
    Rectangle (83,60 42x30), "Ch3", colour toggle: stConnectionDiag.bChannel3
    Rectangle (124,60 42x30), "Ch4", colour toggle: stConnectionDiag.bChannel4
    Rectangle (0,90 166x30), "Diag: %s", text variable: stConnectionDiag.sDiag, colour toggle: stConnectionDiag.sDiag <> 'No error'
    Rectangle (0,120 166x30), "State: %s", text variable: stConnectionDiag.sState
    Rectangle (0,150 83x30), "T1: %s °C", text variable: stConnectionDiag.stSlaveTemp.nInternalTemperature1, colour toggle: stConnectionDiag.bTempWarning
    Rectangle (83,150 83x30), "T2: %s °C", text variable: stConnectionDiag.stSlaveTemp.nInternalTemperature2, colour toggle: stConnectionDiag.bTempWarning
    Rectangle (0,30 166x30), "%s", text variable: stConnectionDiag.sEcSlaveType
    Rectangle (84,81 81x8), "Err input pair", invisible if: NOT stConnectionDiag.stTsDiagObjectsBitsEL1904.bErrSecondInputPair
    Rectangle (1,61 40x8), "Err", invisible if: NOT stConnectionDiag.stTsDiagObjectsBitsEL1904.bErrInput1
    Rectangle (43,61 39x8), "Err", invisible if: NOT stConnectionDiag.stTsDiagObjectsBitsEL1904.bErrInput2
    Rectangle (84,61 39x8), "Err", invisible if: NOT stConnectionDiag.stTsDiagObjectsBitsEL1904.bErrInput3
    Rectangle (125,61 40x8), "Err", invisible if: NOT stConnectionDiag.stTsDiagObjectsBitsEL1904.bErrInput4
    Rectangle (1,81 81x8), "Err input pair", invisible if: NOT stConnectionDiag.stTsDiagObjectsBitsEL1904.bErrFirstInputPair
END_VISUALIZATION

// ---- VISUs/HmiTemplatesTwinSAFE/TplTsConnectionEL2904.TcVIS
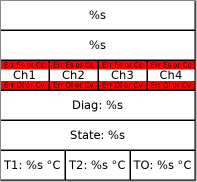
VISUALIZATION TplTsConnectionEL2904  // 197x182
VAR_IN_OUT
	stConnectionDiag 			:FB_TwinSafeConnectionEL2904;
END_VAR
(* End *)
    Rectangle (0,0 195x30), "%s", text variable: stConnectionDiag.sEcSlaveName, colour toggle: stConnectionDiag.sDiag = 'No error'
    Rectangle (0,60 49x30), "Ch1", colour toggle: stConnectionDiag.bChannel1
    Rectangle (49,60 49x30), "Ch2", colour toggle: stConnectionDiag.bChannel2
    Rectangle (98,60 49x30), "Ch3", colour toggle: stConnectionDiag.bChannel3
    Rectangle (147,60 48x30), "Ch4", colour toggle: stConnectionDiag.bChannel4
    Rectangle (0,90 195x30), "Diag: %s", text variable: stConnectionDiag.sDiag, colour toggle: stConnectionDiag.sDiag <> 'No error'
    Rectangle (0,120 195x30), "State: %s", text variable: stConnectionDiag.sState
    Rectangle (0,150 65x30), "T1: %s °C", text variable: stConnectionDiag.stSlaveTemp.nInternalTemperature1, colour toggle: stConnectionDiag.bTempWarning
    Rectangle (65,150 65x30), "T2: %s °C", text variable: stConnectionDiag.stSlaveTemp.nInternalTemperature2, colour toggle: stConnectionDiag.bTempWarning
    Rectangle (0,30 195x30), "%s", text variable: stConnectionDiag.sEcSlaveType
    Rectangle (130,150 65x30), "TO: %s °C", text variable: stConnectionDiag.stSlaveTemp.nInternalTemperatureOutputs, colour toggle: stConnectionDiag.bTempWarning
    Rectangle (148,81 46x8), "Err Ol or Cv", invisible if: NOT stConnectionDiag.stTsDiagObjectsBitsEL2904.bOlOrCvErrOutput4
    Rectangle (148,61 46x8), "Err Es or Cc", invisible if: NOT stConnectionDiag.stTsDiagObjectsBitsEL2904.bEsOrCcErrOutput4
    Rectangle (99,61 47x8), "Err Es or Cc", invisible if: NOT stConnectionDiag.stTsDiagObjectsBitsEL2904.bEsOrCcErrOutput3
    Rectangle (99,81 47x8), "Err Ol or Cv", invisible if: NOT stConnectionDiag.stTsDiagObjectsBitsEL2904.bOlOrCvErrOutput3
    Rectangle (50,61 47x8), "Err Es or Cc", invisible if: NOT stConnectionDiag.stTsDiagObjectsBitsEL2904.bEsOrCcErrOutput2
    Rectangle (50,81 47x8), "Err Ol or Cv", invisible if: NOT stConnectionDiag.stTsDiagObjectsBitsEL2904.bOlOrCvErrOutput2
    Rectangle (1,61 47x8), "Err Es or Cc", invisible if: NOT stConnectionDiag.stTsDiagObjectsBitsEL2904.bEsOrCcErrOutput1
    Rectangle (1,81 47x8), "Err Ol or Cv", invisible if: NOT stConnectionDiag.stTsDiagObjectsBitsEL2904.bOlOrCvErrOutput1
END_VISUALIZATION

// ---- VISUs/HmiTemplatesTwinSAFE/TplTsConnectionEL3214.TcVIS
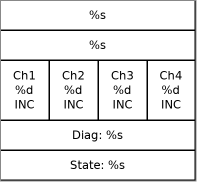
VISUALIZATION TplTsConnectionEL3214  // 197x182
VAR_IN_OUT
	stConnectionDiag 			:FB_TwinSafeConnectionEL3214;
END_VAR
(* End *)
    Rectangle (0,0 195x30), "%s", text variable: stConnectionDiag.sEcSlaveName, colour toggle: stConnectionDiag.sDiag = 'No error'
    Rectangle (0,60 49x60), "Ch1 %d INC", text variable: stConnectionDiag.nInSafeDataValue1
    Rectangle (49,60 49x60), "Ch2 %d INC", text variable: stConnectionDiag.nInSafeDataValue2
    Rectangle (98,60 49x60), "Ch3 %d INC", text variable: stConnectionDiag.nInSafeDataValue3
    Rectangle (147,60 48x60), "Ch4 %d INC", text variable: stConnectionDiag.nInSafeDataValue4
    Rectangle (0,120 195x30), "Diag: %s", text variable: stConnectionDiag.sDiag, colour toggle: stConnectionDiag.sDiag <> 'No error'
    Rectangle (0,150 195x30), "State: %s", text variable: stConnectionDiag.sState
    Rectangle (0,30 195x30), "%s", text variable: stConnectionDiag.sEcSlaveType
END_VISUALIZATION

// ---- VISUs/HmiTemplatesTwinSAFE/TplTsConnectionEL5021.TcVIS
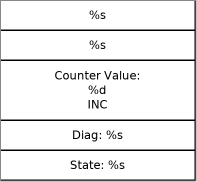
VISUALIZATION TplTsConnectionEL5021  // 197x182
VAR_IN_OUT
	stConnectionDiag 			:FB_TwinSafeConnectionEL5021;
END_VAR
(* End *)
    Rectangle (0,0 195x30), "%s", text variable: stConnectionDiag.sEcSlaveName, colour toggle: stConnectionDiag.sDiag = 'No error'
    Rectangle (0,60 195x60), "Counter Value: %d INC", text variable: stConnectionDiag.nInSafeDataCounterValue
    Rectangle (0,120 195x30), "Diag: %s", text variable: stConnectionDiag.sDiag, colour toggle: stConnectionDiag.sDiag <> 'No error'
    Rectangle (0,150 195x30), "State: %s", text variable: stConnectionDiag.sState
    Rectangle (0,30 195x30), "%s", text variable: stConnectionDiag.sEcSlaveType
END_VISUALIZATION

// ---- VISUs/HmiTemplatesTwinSAFE/TplTsFb.TcVIS
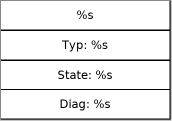
VISUALIZATION TplTsFb  // 172x121
VAR_IN_OUT
	stfbDiag 					:FB_TwinSafeFB;
END_VAR
(* End *)
    Rectangle (0,0 170x30), "%s", text variable: stfbDiag.sName, colour toggle: stfbDiag.sState = 'RUN' or stfbDiag.sState = 'MON_ON'
    Rectangle (0,30 170x30), "Typ: %s", text variable: stfbDiag.sType
    Rectangle (0,60 170x30), "State: %s", text variable: stfbDiag.sState, colour toggle: stfbDiag.sState = 'ERROR'
    Rectangle (0,89 170x30), "Diag: %s", text variable: stfbDiag.sDiag
END_VISUALIZATION

// ---- VISUs/HmiTemplatesTwinSAFE/TplTsGroup.TcVIS
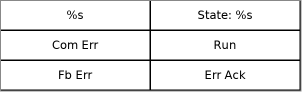
VISUALIZATION TplTsGroup  // 302x92
VAR_IN_OUT
	stGroupDiag					:FB_TwinSafeGroup;
END_VAR
(* End *)
    Rectangle (0,30 150x30), "Com Err", colour toggle: stGroupDiag.bComErr
    Rectangle (0,60 150x30), "Fb Err", colour toggle: stGroupDiag.bFbErr
    Rectangle (150,0 150x30), "State: %s", text variable: stGroupDiag.sState, colour toggle: stGroupDiag.sState = 'ERROR'
    Rectangle (150,30 150x30), "Run", colour toggle: stGroupDiag.bRun
    Rectangle (150,60 150x30), "Err Ack", colour toggle: stGroupDiag.bErrAck
    Rectangle (0,0 150x30), "%s", text variable: stGroupDiag.sName, colour toggle: stGroupDiag.sState = 'RUN'
END_VISUALIZATION

// ---- VISUs/HmiTemplatesTwinSAFE/TplTsGroupExt.TcVIS
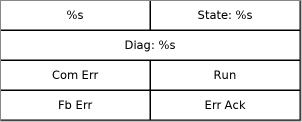
VISUALIZATION TplTsGroupExt  // 302x122
VAR_IN_OUT
	stGroupDiag					:FB_TwinSafeGroupExt;
END_VAR
(* End *)
    Rectangle (0,60 150x30), "Com Err", colour toggle: stGroupDiag.bComErr
    Rectangle (0,90 150x30), "Fb Err", colour toggle: stGroupDiag.bFbErr
    Rectangle (150,0 150x30), "State: %s", text variable: stGroupDiag.sState, colour toggle: stGroupDiag.sState = 'ERROR'
    Rectangle (150,60 150x30), "Run", colour toggle: stGroupDiag.bRun
    Rectangle (150,90 150x30), "Err Ack", colour toggle: stGroupDiag.bErrAck
    Rectangle (0,0 150x30), "%s", text variable: stGroupDiag.sName, colour toggle: stGroupDiag.sState = 'RUN'
    Rectangle (0,30 300x30), "Diag: %s", text variable: stGroupDiag.sDiag
END_VISUALIZATION

// ---- VISUs/HmiTwinSAFEDiagnostic.TcVIS
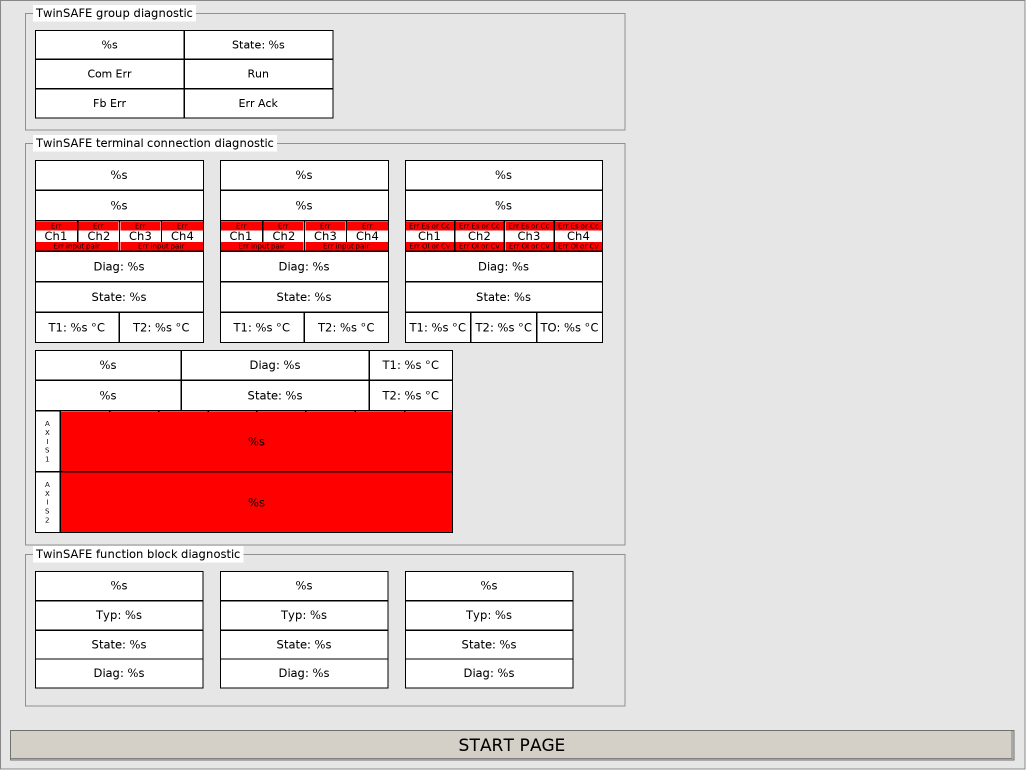
VISUALIZATION HmiTwinSAFEDiagnostic  // 1026x770
    Rectangle (0,0 1024x768)
    GroupBox (25,5 600x125), "TwinSAFE group diagnostic"
        Frame (10,25 300x90)
            shows TplTsGroup(stGroupDiag := TwinSAFE.fbSafeGroup1)
    GroupBox (25,135 600x410), "TwinSAFE terminal connection diagnostic"
        Frame (195,25 171x185)
            shows TplTsConnectionEL1904(stConnectionDiag := TwinSAFE.fbSafeConnectionEL1904_2_Group1)
        Frame (380,25 200x185)
            shows TplTsConnectionEL2904(stConnectionDiag := TwinSAFE.fbSafeConnectionEL2904_1_Group1)
        Frame (10,25 171x185)
            shows TplTsConnectionEL1904(stConnectionDiag := TwinSAFE.fbSafeConnectionEL1904_1_Group1)
        Frame (10,215 420x185)
            shows TplTsConnectionAX5805(stConnectionDiag := TwinSAFE.fbSafeConnectionAX5805_1_Group1)
    GroupBox (25,546 600x160), "TwinSAFE function block diagnostic"
        Frame (10,25 170x119)
            shows TplTsFb(stfbDiag := TwinSAFE.fbSafeFB_1_Group1)
        Frame (195,25 170x119)
            shows TplTsFb(stfbDiag := TwinSAFE.fbSafeFB_2_Group1)
        Frame (380,25 170x119)
            shows TplTsFb(stfbDiag := TwinSAFE.fbSafeFB_3_Group1)
    Button (10,730 1004x30), "START PAGE"
        OnMouseClick: change screen: HmiStartPage
END_VISUALIZATION
